{attribute 'linkalways'} 
{attribute 'no_explicit_call' := 'This FB is a CLASS and must be accessed using methods or properties'}
{attribute 'enable_dynamic_creation'}
FUNCTION_BLOCK CollectionNode IMPLEMENTS I_CollectionNode
VAR
	collectableObject : I_Collectable;
	nextNode : I_CollectionNode;
END_VAR

PROPERTY PUBLIC Collectable : I_Collectable
GET
collectable := collectableObject;
END_GET
END_PROPERTY

METHOD PUBLIC Destroy
VAR_INPUT
END_VAR
__DELETE(THIS);
END_METHOD

METHOD FB_init : BOOL
VAR_INPUT
	bInitRetains : BOOL; // if TRUE, the retain variables are initialized (warm start / cold start)
	bInCopyCode : BOOL;  // if TRUE, the instance afterwards gets moved into the copy code (online change)
	Collectable : I_Collectable;
END_VAR
collectableObject := Collectable;
END_METHOD

PROPERTY PUBLIC Next : I_CollectionNode
GET
Next := nextNode;
END_GET
SET // PUBLIC
nextNode := Next;
END_SET
END_PROPERTY

END_FUNCTION_BLOCK

(* stored: Version 1.1.0.1, ProductVersion 3.1.4024.12
   POU CollectionNode: Id {5adfdc88-b543-015b-2e2d-e93d2ecab915}, SpecialFunc None
   Folder Constructor: Id {a1b45c4d-9f03-09ac-3f57-cbd76a7b8021}
   Property Collectable: Id {6c311c39-3df1-0be4-2859-1f08eb7a73a7}
   Get Get: Id {a12447c9-70a9-07ac-1d7a-cebc691d7dde}
   Method Destroy: Id {c2f88645-62f4-0f40-0a08-0489d1ba0e29}
   Method FB_init: Id {867a08eb-acb7-0f4e-0543-703e7f2f3578}
   Property Next: Id {1ef045eb-e80f-0b1e-09f6-13565fd4e6ee}
   Get Get: Id {d62389ff-2028-0ef9-36a8-a499e84e1ee9}
   Set Set: Id {6241b4ad-71c1-0b69-2c09-f02ce1c75c5f} *)
